GLOBALCONSTANTS SoftKeyActivationCode (* SoftKeyActivationCode constants *)
  (* Standard: 61499-1; Description: Copyright (c) 2024 HR Agrartechnik GmbH This program and the accompanying materials are made available under the terms of the Eclipse Public License 2.0 which is available at https://www.eclipse.org/legal/epl-2.0/ SPDX-License-Identifier: EPL-2.0 *)
  (* Version 1.0, 2024-01-25, Franz Höpfinger, HR Agrartechnik GmbH *)
  VAR_GLOBAL CONSTANT
    SK_RELEASED : SoftKeyActivationCode_S := (code := 0); (* SoftKey has been released (state change) *)
    SK_PRESSED : SoftKeyActivationCode_S := (code := 1); (* SoftKey  has been pressed (state change) *)
    SK_STILL_HELD : SoftKeyActivationCode_S := (code := 2); (* SoftKey is still held *)
    SK_ABORTED : SoftKeyActivationCode_S := (code := 3); (* SoftKey press aborted (Applies to VT version 4 and later) *)
    Invalid : SoftKeyActivationCode_S := (code := 255);
  END_VAR
END_GLOBALCONSTANTS
